PROGRAM MAIN
VAR
END_VAR

Delta_Robot_Program();

END_PROGRAM

(* stored: Version 1.1.0.1, ProductVersion 3.1.4024.12
   POU MAIN: Id {d93ec619-9daf-4e08-ad99-c2277f7176e2}, SpecialFunc None *)
